// TIA Portal V21 export
FUNCTION "PHT_ValveLogic" : Void   // FC1207, LAD
{ S7_Optimized_Access := 'TRUE' }
// stored: AutoNumber false, SetENOAutomatically false
BEGIN

REGION Network 1: ________________________________LINE VALVE________________________________
END_REGION

REGION Network 2: "PhtCycle".Cv24 - CAI
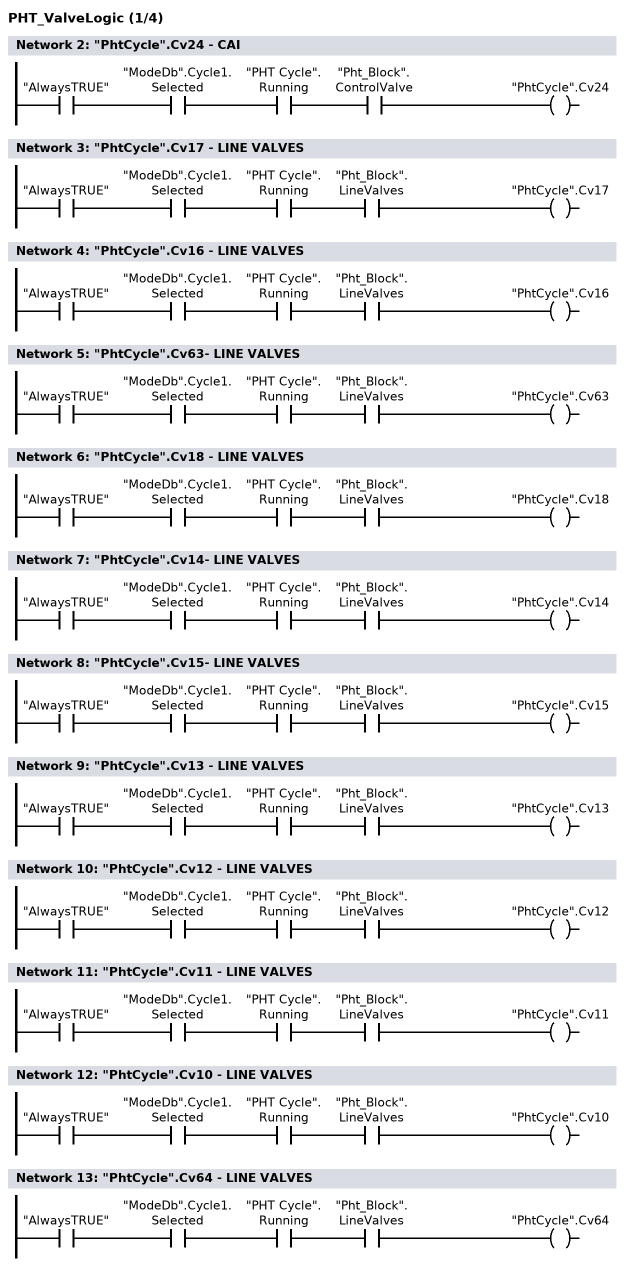
   RUNG wire#powerrail
      Contact( "AlwaysTRUE" )
      Contact( "ModeDb".Cycle1.Selected )
      Contact( "PHT Cycle".Running )
      Contact( "Pht_Block".ControlValve )
      Coil( "PhtCycle".Cv24 )
   END_RUNG
   // the same network as SCL:
   "PhtCycle".Cv24 := "AlwaysTRUE" AND "ModeDb".Cycle1.Selected AND "PHT Cycle".Running AND "Pht_Block".ControlValve;
END_REGION

REGION Network 3: "PhtCycle".Cv17 - LINE VALVES
   RUNG wire#powerrail
      Contact( "AlwaysTRUE" )
      Contact( "ModeDb".Cycle1.Selected )
      Contact( "PHT Cycle".Running )
      Contact( "Pht_Block".LineValves )
      Coil( "PhtCycle".Cv17 )
   END_RUNG
   // the same network as SCL:
   "PhtCycle".Cv17 := "AlwaysTRUE" AND "ModeDb".Cycle1.Selected AND "PHT Cycle".Running AND "Pht_Block".LineValves;
END_REGION

REGION Network 4: "PhtCycle".Cv16 - LINE VALVES
   RUNG wire#powerrail
      Contact( "AlwaysTRUE" )
      Contact( "ModeDb".Cycle1.Selected )
      Contact( "PHT Cycle".Running )
      Contact( "Pht_Block".LineValves )
      Coil( "PhtCycle".Cv16 )
   END_RUNG
   // the same network as SCL:
   "PhtCycle".Cv16 := "AlwaysTRUE" AND "ModeDb".Cycle1.Selected AND "PHT Cycle".Running AND "Pht_Block".LineValves;
END_REGION

REGION Network 5: "PhtCycle".Cv63- LINE VALVES
   RUNG wire#powerrail
      Contact( "AlwaysTRUE" )
      Contact( "ModeDb".Cycle1.Selected )
      Contact( "PHT Cycle".Running )
      Contact( "Pht_Block".LineValves )
      Coil( "PhtCycle".Cv63 )
   END_RUNG
   // the same network as SCL:
   "PhtCycle".Cv63 := "AlwaysTRUE" AND "ModeDb".Cycle1.Selected AND "PHT Cycle".Running AND "Pht_Block".LineValves;
END_REGION

REGION Network 6: "PhtCycle".Cv18 - LINE VALVES
   RUNG wire#powerrail
      Contact( "AlwaysTRUE" )
      Contact( "ModeDb".Cycle1.Selected )
      Contact( "PHT Cycle".Running )
      Contact( "Pht_Block".LineValves )
      Coil( "PhtCycle".Cv18 )
   END_RUNG
   // the same network as SCL:
   "PhtCycle".Cv18 := "AlwaysTRUE" AND "ModeDb".Cycle1.Selected AND "PHT Cycle".Running AND "Pht_Block".LineValves;
END_REGION

REGION Network 7: "PhtCycle".Cv14- LINE VALVES
   RUNG wire#powerrail
      Contact( "AlwaysTRUE" )
      Contact( "ModeDb".Cycle1.Selected )
      Contact( "PHT Cycle".Running )
      Contact( "Pht_Block".LineValves )
      Coil( "PhtCycle".Cv14 )
   END_RUNG
   // the same network as SCL:
   "PhtCycle".Cv14 := "AlwaysTRUE" AND "ModeDb".Cycle1.Selected AND "PHT Cycle".Running AND "Pht_Block".LineValves;
END_REGION

REGION Network 8: "PhtCycle".Cv15- LINE VALVES
   RUNG wire#powerrail
      Contact( "AlwaysTRUE" )
      Contact( "ModeDb".Cycle1.Selected )
      Contact( "PHT Cycle".Running )
      Contact( "Pht_Block".LineValves )
      Coil( "PhtCycle".Cv15 )
   END_RUNG
   // the same network as SCL:
   "PhtCycle".Cv15 := "AlwaysTRUE" AND "ModeDb".Cycle1.Selected AND "PHT Cycle".Running AND "Pht_Block".LineValves;
END_REGION

REGION Network 9: "PhtCycle".Cv13 - LINE VALVES
   RUNG wire#powerrail
      Contact( "AlwaysTRUE" )
      Contact( "ModeDb".Cycle1.Selected )
      Contact( "PHT Cycle".Running )
      Contact( "Pht_Block".LineValves )
      Coil( "PhtCycle".Cv13 )
   END_RUNG
   // the same network as SCL:
   "PhtCycle".Cv13 := "AlwaysTRUE" AND "ModeDb".Cycle1.Selected AND "PHT Cycle".Running AND "Pht_Block".LineValves;
END_REGION

REGION Network 10: "PhtCycle".Cv12 - LINE VALVES
   RUNG wire#powerrail
      Contact( "AlwaysTRUE" )
      Contact( "ModeDb".Cycle1.Selected )
      Contact( "PHT Cycle".Running )
      Contact( "Pht_Block".LineValves )
      Coil( "PhtCycle".Cv12 )
   END_RUNG
   // the same network as SCL:
   "PhtCycle".Cv12 := "AlwaysTRUE" AND "ModeDb".Cycle1.Selected AND "PHT Cycle".Running AND "Pht_Block".LineValves;
END_REGION

REGION Network 11: "PhtCycle".Cv11 - LINE VALVES
   RUNG wire#powerrail
      Contact( "AlwaysTRUE" )
      Contact( "ModeDb".Cycle1.Selected )
      Contact( "PHT Cycle".Running )
      Contact( "Pht_Block".LineValves )
      Coil( "PhtCycle".Cv11 )
   END_RUNG
   // the same network as SCL:
   "PhtCycle".Cv11 := "AlwaysTRUE" AND "ModeDb".Cycle1.Selected AND "PHT Cycle".Running AND "Pht_Block".LineValves;
END_REGION

REGION Network 12: "PhtCycle".Cv10 - LINE VALVES
   RUNG wire#powerrail
      Contact( "AlwaysTRUE" )
      Contact( "ModeDb".Cycle1.Selected )
      Contact( "PHT Cycle".Running )
      Contact( "Pht_Block".LineValves )
      Coil( "PhtCycle".Cv10 )
   END_RUNG
   // the same network as SCL:
   "PhtCycle".Cv10 := "AlwaysTRUE" AND "ModeDb".Cycle1.Selected AND "PHT Cycle".Running AND "Pht_Block".LineValves;
END_REGION

REGION Network 13: "PhtCycle".Cv64 - LINE VALVES
   RUNG wire#powerrail
      Contact( "AlwaysTRUE" )
      Contact( "ModeDb".Cycle1.Selected )
      Contact( "PHT Cycle".Running )
      Contact( "Pht_Block".LineValves )
      Coil( "PhtCycle".Cv64 )
   END_RUNG
   // the same network as SCL:
   "PhtCycle".Cv64 := "AlwaysTRUE" AND "ModeDb".Cycle1.Selected AND "PHT Cycle".Running AND "Pht_Block".LineValves;
END_REGION

REGION Network 14: "PhtCycle".Cv26 - LINE VALVES
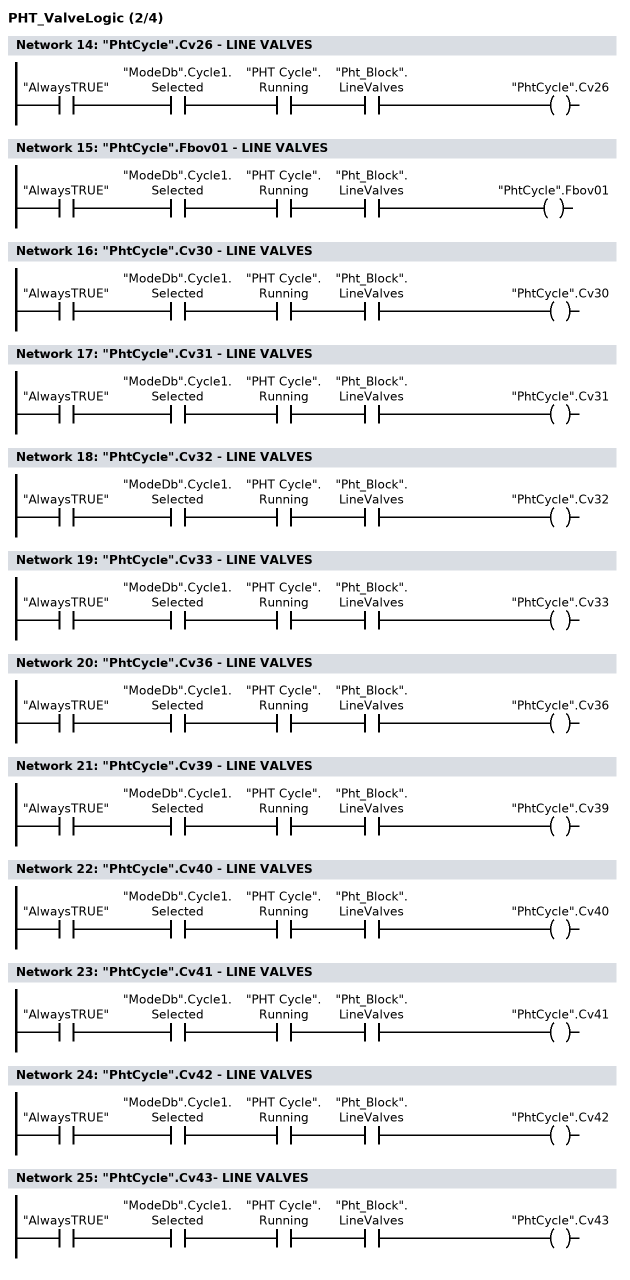
   RUNG wire#powerrail
      Contact( "AlwaysTRUE" )
      Contact( "ModeDb".Cycle1.Selected )
      Contact( "PHT Cycle".Running )
      Contact( "Pht_Block".LineValves )
      Coil( "PhtCycle".Cv26 )
   END_RUNG
   // the same network as SCL:
   "PhtCycle".Cv26 := "AlwaysTRUE" AND "ModeDb".Cycle1.Selected AND "PHT Cycle".Running AND "Pht_Block".LineValves;
END_REGION

REGION Network 15: "PhtCycle".Fbov01 - LINE VALVES
   RUNG wire#powerrail
      Contact( "AlwaysTRUE" )
      Contact( "ModeDb".Cycle1.Selected )
      Contact( "PHT Cycle".Running )
      Contact( "Pht_Block".LineValves )
      Coil( "PhtCycle".Fbov01 )
   END_RUNG
   // the same network as SCL:
   "PhtCycle".Fbov01 := "AlwaysTRUE" AND "ModeDb".Cycle1.Selected AND "PHT Cycle".Running AND "Pht_Block".LineValves;
END_REGION

REGION Network 16: "PhtCycle".Cv30 - LINE VALVES
   RUNG wire#powerrail
      Contact( "AlwaysTRUE" )
      Contact( "ModeDb".Cycle1.Selected )
      Contact( "PHT Cycle".Running )
      Contact( "Pht_Block".LineValves )
      Coil( "PhtCycle".Cv30 )
   END_RUNG
   // the same network as SCL:
   "PhtCycle".Cv30 := "AlwaysTRUE" AND "ModeDb".Cycle1.Selected AND "PHT Cycle".Running AND "Pht_Block".LineValves;
END_REGION

REGION Network 17: "PhtCycle".Cv31 - LINE VALVES
   RUNG wire#powerrail
      Contact( "AlwaysTRUE" )
      Contact( "ModeDb".Cycle1.Selected )
      Contact( "PHT Cycle".Running )
      Contact( "Pht_Block".LineValves )
      Coil( "PhtCycle".Cv31 )
   END_RUNG
   // the same network as SCL:
   "PhtCycle".Cv31 := "AlwaysTRUE" AND "ModeDb".Cycle1.Selected AND "PHT Cycle".Running AND "Pht_Block".LineValves;
END_REGION

REGION Network 18: "PhtCycle".Cv32 - LINE VALVES
   RUNG wire#powerrail
      Contact( "AlwaysTRUE" )
      Contact( "ModeDb".Cycle1.Selected )
      Contact( "PHT Cycle".Running )
      Contact( "Pht_Block".LineValves )
      Coil( "PhtCycle".Cv32 )
   END_RUNG
   // the same network as SCL:
   "PhtCycle".Cv32 := "AlwaysTRUE" AND "ModeDb".Cycle1.Selected AND "PHT Cycle".Running AND "Pht_Block".LineValves;
END_REGION

REGION Network 19: "PhtCycle".Cv33 - LINE VALVES
   RUNG wire#powerrail
      Contact( "AlwaysTRUE" )
      Contact( "ModeDb".Cycle1.Selected )
      Contact( "PHT Cycle".Running )
      Contact( "Pht_Block".LineValves )
      Coil( "PhtCycle".Cv33 )
   END_RUNG
   // the same network as SCL:
   "PhtCycle".Cv33 := "AlwaysTRUE" AND "ModeDb".Cycle1.Selected AND "PHT Cycle".Running AND "Pht_Block".LineValves;
END_REGION

REGION Network 20: "PhtCycle".Cv36 - LINE VALVES
   RUNG wire#powerrail
      Contact( "AlwaysTRUE" )
      Contact( "ModeDb".Cycle1.Selected )
      Contact( "PHT Cycle".Running )
      Contact( "Pht_Block".LineValves )
      Coil( "PhtCycle".Cv36 )
   END_RUNG
   // the same network as SCL:
   "PhtCycle".Cv36 := "AlwaysTRUE" AND "ModeDb".Cycle1.Selected AND "PHT Cycle".Running AND "Pht_Block".LineValves;
END_REGION

REGION Network 21: "PhtCycle".Cv39 - LINE VALVES
   RUNG wire#powerrail
      Contact( "AlwaysTRUE" )
      Contact( "ModeDb".Cycle1.Selected )
      Contact( "PHT Cycle".Running )
      Contact( "Pht_Block".LineValves )
      Coil( "PhtCycle".Cv39 )
   END_RUNG
   // the same network as SCL:
   "PhtCycle".Cv39 := "AlwaysTRUE" AND "ModeDb".Cycle1.Selected AND "PHT Cycle".Running AND "Pht_Block".LineValves;
END_REGION

REGION Network 22: "PhtCycle".Cv40 - LINE VALVES
   RUNG wire#powerrail
      Contact( "AlwaysTRUE" )
      Contact( "ModeDb".Cycle1.Selected )
      Contact( "PHT Cycle".Running )
      Contact( "Pht_Block".LineValves )
      Coil( "PhtCycle".Cv40 )
   END_RUNG
   // the same network as SCL:
   "PhtCycle".Cv40 := "AlwaysTRUE" AND "ModeDb".Cycle1.Selected AND "PHT Cycle".Running AND "Pht_Block".LineValves;
END_REGION

REGION Network 23: "PhtCycle".Cv41 - LINE VALVES
   RUNG wire#powerrail
      Contact( "AlwaysTRUE" )
      Contact( "ModeDb".Cycle1.Selected )
      Contact( "PHT Cycle".Running )
      Contact( "Pht_Block".LineValves )
      Coil( "PhtCycle".Cv41 )
   END_RUNG
   // the same network as SCL:
   "PhtCycle".Cv41 := "AlwaysTRUE" AND "ModeDb".Cycle1.Selected AND "PHT Cycle".Running AND "Pht_Block".LineValves;
END_REGION

REGION Network 24: "PhtCycle".Cv42 - LINE VALVES
   RUNG wire#powerrail
      Contact( "AlwaysTRUE" )
      Contact( "ModeDb".Cycle1.Selected )
      Contact( "PHT Cycle".Running )
      Contact( "Pht_Block".LineValves )
      Coil( "PhtCycle".Cv42 )
   END_RUNG
   // the same network as SCL:
   "PhtCycle".Cv42 := "AlwaysTRUE" AND "ModeDb".Cycle1.Selected AND "PHT Cycle".Running AND "Pht_Block".LineValves;
END_REGION

REGION Network 25: "PhtCycle".Cv43- LINE VALVES
   RUNG wire#powerrail
      Contact( "AlwaysTRUE" )
      Contact( "ModeDb".Cycle1.Selected )
      Contact( "PHT Cycle".Running )
      Contact( "Pht_Block".LineValves )
      Coil( "PhtCycle".Cv43 )
   END_RUNG
   // the same network as SCL:
   "PhtCycle".Cv43 := "AlwaysTRUE" AND "ModeDb".Cycle1.Selected AND "PHT Cycle".Running AND "Pht_Block".LineValves;
END_REGION

REGION Network 26: "PhtCycle".Cv44 - LINE VALVES
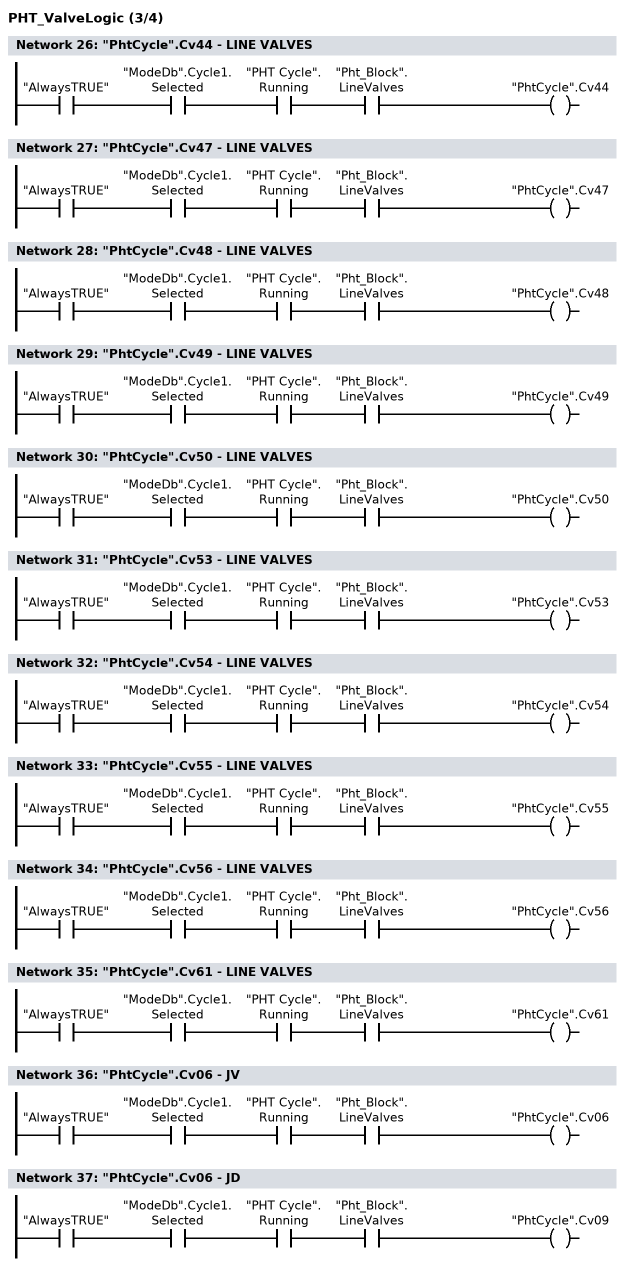
   RUNG wire#powerrail
      Contact( "AlwaysTRUE" )
      Contact( "ModeDb".Cycle1.Selected )
      Contact( "PHT Cycle".Running )
      Contact( "Pht_Block".LineValves )
      Coil( "PhtCycle".Cv44 )
   END_RUNG
   // the same network as SCL:
   "PhtCycle".Cv44 := "AlwaysTRUE" AND "ModeDb".Cycle1.Selected AND "PHT Cycle".Running AND "Pht_Block".LineValves;
END_REGION

REGION Network 27: "PhtCycle".Cv47 - LINE VALVES
   RUNG wire#powerrail
      Contact( "AlwaysTRUE" )
      Contact( "ModeDb".Cycle1.Selected )
      Contact( "PHT Cycle".Running )
      Contact( "Pht_Block".LineValves )
      Coil( "PhtCycle".Cv47 )
   END_RUNG
   // the same network as SCL:
   "PhtCycle".Cv47 := "AlwaysTRUE" AND "ModeDb".Cycle1.Selected AND "PHT Cycle".Running AND "Pht_Block".LineValves;
END_REGION

REGION Network 28: "PhtCycle".Cv48 - LINE VALVES
   RUNG wire#powerrail
      Contact( "AlwaysTRUE" )
      Contact( "ModeDb".Cycle1.Selected )
      Contact( "PHT Cycle".Running )
      Contact( "Pht_Block".LineValves )
      Coil( "PhtCycle".Cv48 )
   END_RUNG
   // the same network as SCL:
   "PhtCycle".Cv48 := "AlwaysTRUE" AND "ModeDb".Cycle1.Selected AND "PHT Cycle".Running AND "Pht_Block".LineValves;
END_REGION

REGION Network 29: "PhtCycle".Cv49 - LINE VALVES
   RUNG wire#powerrail
      Contact( "AlwaysTRUE" )
      Contact( "ModeDb".Cycle1.Selected )
      Contact( "PHT Cycle".Running )
      Contact( "Pht_Block".LineValves )
      Coil( "PhtCycle".Cv49 )
   END_RUNG
   // the same network as SCL:
   "PhtCycle".Cv49 := "AlwaysTRUE" AND "ModeDb".Cycle1.Selected AND "PHT Cycle".Running AND "Pht_Block".LineValves;
END_REGION

REGION Network 30: "PhtCycle".Cv50 - LINE VALVES
   RUNG wire#powerrail
      Contact( "AlwaysTRUE" )
      Contact( "ModeDb".Cycle1.Selected )
      Contact( "PHT Cycle".Running )
      Contact( "Pht_Block".LineValves )
      Coil( "PhtCycle".Cv50 )
   END_RUNG
   // the same network as SCL:
   "PhtCycle".Cv50 := "AlwaysTRUE" AND "ModeDb".Cycle1.Selected AND "PHT Cycle".Running AND "Pht_Block".LineValves;
END_REGION

REGION Network 31: "PhtCycle".Cv53 - LINE VALVES
   RUNG wire#powerrail
      Contact( "AlwaysTRUE" )
      Contact( "ModeDb".Cycle1.Selected )
      Contact( "PHT Cycle".Running )
      Contact( "Pht_Block".LineValves )
      Coil( "PhtCycle".Cv53 )
   END_RUNG
   // the same network as SCL:
   "PhtCycle".Cv53 := "AlwaysTRUE" AND "ModeDb".Cycle1.Selected AND "PHT Cycle".Running AND "Pht_Block".LineValves;
END_REGION

REGION Network 32: "PhtCycle".Cv54 - LINE VALVES
   RUNG wire#powerrail
      Contact( "AlwaysTRUE" )
      Contact( "ModeDb".Cycle1.Selected )
      Contact( "PHT Cycle".Running )
      Contact( "Pht_Block".LineValves )
      Coil( "PhtCycle".Cv54 )
   END_RUNG
   // the same network as SCL:
   "PhtCycle".Cv54 := "AlwaysTRUE" AND "ModeDb".Cycle1.Selected AND "PHT Cycle".Running AND "Pht_Block".LineValves;
END_REGION

REGION Network 33: "PhtCycle".Cv55 - LINE VALVES
   RUNG wire#powerrail
      Contact( "AlwaysTRUE" )
      Contact( "ModeDb".Cycle1.Selected )
      Contact( "PHT Cycle".Running )
      Contact( "Pht_Block".LineValves )
      Coil( "PhtCycle".Cv55 )
   END_RUNG
   // the same network as SCL:
   "PhtCycle".Cv55 := "AlwaysTRUE" AND "ModeDb".Cycle1.Selected AND "PHT Cycle".Running AND "Pht_Block".LineValves;
END_REGION

REGION Network 34: "PhtCycle".Cv56 - LINE VALVES
   RUNG wire#powerrail
      Contact( "AlwaysTRUE" )
      Contact( "ModeDb".Cycle1.Selected )
      Contact( "PHT Cycle".Running )
      Contact( "Pht_Block".LineValves )
      Coil( "PhtCycle".Cv56 )
   END_RUNG
   // the same network as SCL:
   "PhtCycle".Cv56 := "AlwaysTRUE" AND "ModeDb".Cycle1.Selected AND "PHT Cycle".Running AND "Pht_Block".LineValves;
END_REGION

REGION Network 35: "PhtCycle".Cv61 - LINE VALVES
   RUNG wire#powerrail
      Contact( "AlwaysTRUE" )
      Contact( "ModeDb".Cycle1.Selected )
      Contact( "PHT Cycle".Running )
      Contact( "Pht_Block".LineValves )
      Coil( "PhtCycle".Cv61 )
   END_RUNG
   // the same network as SCL:
   "PhtCycle".Cv61 := "AlwaysTRUE" AND "ModeDb".Cycle1.Selected AND "PHT Cycle".Running AND "Pht_Block".LineValves;
END_REGION

REGION Network 36: "PhtCycle".Cv06 - JV
   RUNG wire#powerrail
      Contact( "AlwaysTRUE" )
      Contact( "ModeDb".Cycle1.Selected )
      Contact( "PHT Cycle".Running )
      Contact( "Pht_Block".LineValves )
      Coil( "PhtCycle".Cv06 )
   END_RUNG
   // the same network as SCL:
   "PhtCycle".Cv06 := "AlwaysTRUE" AND "ModeDb".Cycle1.Selected AND "PHT Cycle".Running AND "Pht_Block".LineValves;
END_REGION

REGION Network 37: "PhtCycle".Cv06 - JD
   RUNG wire#powerrail
      Contact( "AlwaysTRUE" )
      Contact( "ModeDb".Cycle1.Selected )
      Contact( "PHT Cycle".Running )
      Contact( "Pht_Block".LineValves )
      Coil( "PhtCycle".Cv09 )
   END_RUNG
   // the same network as SCL:
   "PhtCycle".Cv09 := "AlwaysTRUE" AND "ModeDb".Cycle1.Selected AND "PHT Cycle".Running AND "Pht_Block".LineValves;
END_REGION

REGION Network 38: ________________________________RELEASE VALVE________________________________
END_REGION

REGION Network 39: "PhtCycle".Cv25 - RELEASE VALVE
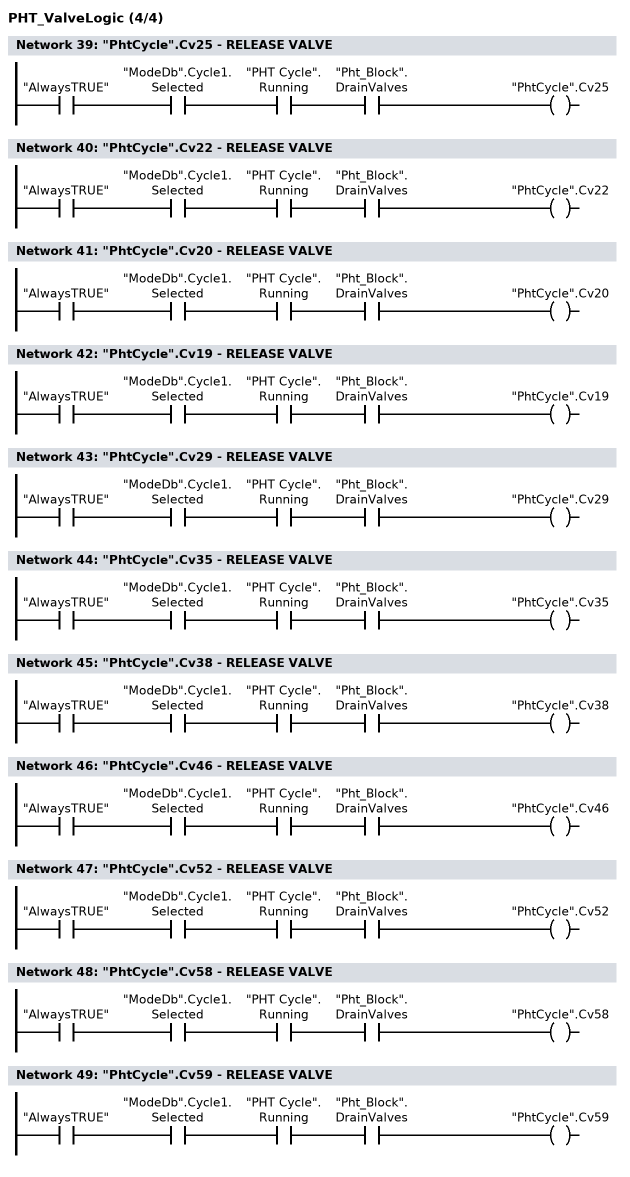
   RUNG wire#powerrail
      Contact( "AlwaysTRUE" )
      Contact( "ModeDb".Cycle1.Selected )
      Contact( "PHT Cycle".Running )
      Contact( "Pht_Block".DrainValves )
      Coil( "PhtCycle".Cv25 )
   END_RUNG
   // the same network as SCL:
   "PhtCycle".Cv25 := "AlwaysTRUE" AND "ModeDb".Cycle1.Selected AND "PHT Cycle".Running AND "Pht_Block".DrainValves;
END_REGION

REGION Network 40: "PhtCycle".Cv22 - RELEASE VALVE
   RUNG wire#powerrail
      Contact( "AlwaysTRUE" )
      Contact( "ModeDb".Cycle1.Selected )
      Contact( "PHT Cycle".Running )
      Contact( "Pht_Block".DrainValves )
      Coil( "PhtCycle".Cv22 )
   END_RUNG
   // the same network as SCL:
   "PhtCycle".Cv22 := "AlwaysTRUE" AND "ModeDb".Cycle1.Selected AND "PHT Cycle".Running AND "Pht_Block".DrainValves;
END_REGION

REGION Network 41: "PhtCycle".Cv20 - RELEASE VALVE
   RUNG wire#powerrail
      Contact( "AlwaysTRUE" )
      Contact( "ModeDb".Cycle1.Selected )
      Contact( "PHT Cycle".Running )
      Contact( "Pht_Block".DrainValves )
      Coil( "PhtCycle".Cv20 )
   END_RUNG
   // the same network as SCL:
   "PhtCycle".Cv20 := "AlwaysTRUE" AND "ModeDb".Cycle1.Selected AND "PHT Cycle".Running AND "Pht_Block".DrainValves;
END_REGION

REGION Network 42: "PhtCycle".Cv19 - RELEASE VALVE
   RUNG wire#powerrail
      Contact( "AlwaysTRUE" )
      Contact( "ModeDb".Cycle1.Selected )
      Contact( "PHT Cycle".Running )
      Contact( "Pht_Block".DrainValves )
      Coil( "PhtCycle".Cv19 )
   END_RUNG
   // the same network as SCL:
   "PhtCycle".Cv19 := "AlwaysTRUE" AND "ModeDb".Cycle1.Selected AND "PHT Cycle".Running AND "Pht_Block".DrainValves;
END_REGION

REGION Network 43: "PhtCycle".Cv29 - RELEASE VALVE
   RUNG wire#powerrail
      Contact( "AlwaysTRUE" )
      Contact( "ModeDb".Cycle1.Selected )
      Contact( "PHT Cycle".Running )
      Contact( "Pht_Block".DrainValves )
      Coil( "PhtCycle".Cv29 )
   END_RUNG
   // the same network as SCL:
   "PhtCycle".Cv29 := "AlwaysTRUE" AND "ModeDb".Cycle1.Selected AND "PHT Cycle".Running AND "Pht_Block".DrainValves;
END_REGION

REGION Network 44: "PhtCycle".Cv35 - RELEASE VALVE
   RUNG wire#powerrail
      Contact( "AlwaysTRUE" )
      Contact( "ModeDb".Cycle1.Selected )
      Contact( "PHT Cycle".Running )
      Contact( "Pht_Block".DrainValves )
      Coil( "PhtCycle".Cv35 )
   END_RUNG
   // the same network as SCL:
   "PhtCycle".Cv35 := "AlwaysTRUE" AND "ModeDb".Cycle1.Selected AND "PHT Cycle".Running AND "Pht_Block".DrainValves;
END_REGION

REGION Network 45: "PhtCycle".Cv38 - RELEASE VALVE
   RUNG wire#powerrail
      Contact( "AlwaysTRUE" )
      Contact( "ModeDb".Cycle1.Selected )
      Contact( "PHT Cycle".Running )
      Contact( "Pht_Block".DrainValves )
      Coil( "PhtCycle".Cv38 )
   END_RUNG
   // the same network as SCL:
   "PhtCycle".Cv38 := "AlwaysTRUE" AND "ModeDb".Cycle1.Selected AND "PHT Cycle".Running AND "Pht_Block".DrainValves;
END_REGION

REGION Network 46: "PhtCycle".Cv46 - RELEASE VALVE
   RUNG wire#powerrail
      Contact( "AlwaysTRUE" )
      Contact( "ModeDb".Cycle1.Selected )
      Contact( "PHT Cycle".Running )
      Contact( "Pht_Block".DrainValves )
      Coil( "PhtCycle".Cv46 )
   END_RUNG
   // the same network as SCL:
   "PhtCycle".Cv46 := "AlwaysTRUE" AND "ModeDb".Cycle1.Selected AND "PHT Cycle".Running AND "Pht_Block".DrainValves;
END_REGION

REGION Network 47: "PhtCycle".Cv52 - RELEASE VALVE
   RUNG wire#powerrail
      Contact( "AlwaysTRUE" )
      Contact( "ModeDb".Cycle1.Selected )
      Contact( "PHT Cycle".Running )
      Contact( "Pht_Block".DrainValves )
      Coil( "PhtCycle".Cv52 )
   END_RUNG
   // the same network as SCL:
   "PhtCycle".Cv52 := "AlwaysTRUE" AND "ModeDb".Cycle1.Selected AND "PHT Cycle".Running AND "Pht_Block".DrainValves;
END_REGION

REGION Network 48: "PhtCycle".Cv58 - RELEASE VALVE
   RUNG wire#powerrail
      Contact( "AlwaysTRUE" )
      Contact( "ModeDb".Cycle1.Selected )
      Contact( "PHT Cycle".Running )
      Contact( "Pht_Block".DrainValves )
      Coil( "PhtCycle".Cv58 )
   END_RUNG
   // the same network as SCL:
   "PhtCycle".Cv58 := "AlwaysTRUE" AND "ModeDb".Cycle1.Selected AND "PHT Cycle".Running AND "Pht_Block".DrainValves;
END_REGION

REGION Network 49: "PhtCycle".Cv59 - RELEASE VALVE
   RUNG wire#powerrail
      Contact( "AlwaysTRUE" )
      Contact( "ModeDb".Cycle1.Selected )
      Contact( "PHT Cycle".Running )
      Contact( "Pht_Block".DrainValves )
      Coil( "PhtCycle".Cv59 )
   END_RUNG
   // the same network as SCL:
   "PhtCycle".Cv59 := "AlwaysTRUE" AND "ModeDb".Cycle1.Selected AND "PHT Cycle".Running AND "Pht_Block".DrainValves;
END_REGION
END_FUNCTION
